(*
SPDX-FileCopyrightText: © 2026 Oleksandr Tiutyk <trofimich@gmail.com>
SPDX-License-Identifier: MIT
License: https://opensource.org/license/mit
*)

(*!
<summary>Exposes the compiler-initialized namespace of the Core library.</summary>
<description>Static internal storage; Name is a borrowed read-only view and requires no cyclic execution.</description>
*)

{attribute 'no_explicit_call' := 'do not call this POU directly'}
PROGRAM INTERNAL CurrentNamespace
VAR
	{attribute 'hide'} 
	_NamespaceExtractor : NamespaceExtractor;
END_VAR

(*!
<summary>Returns the compiler-initialized library namespace.</summary>
<description>Borrowed read-only reference to static storage. Do not modify it through the reference.</description>
*)
{attribute 'monitoring' := 'call'}
PROPERTY Name : REFERENCE TO STRING
GET
Name REF= _NamespaceExtractor.CurrentNamespace;
END_GET
END_PROPERTY

END_PROGRAM

(* stored: Version 1.1.0.1
   POU CurrentNamespace: Id {d326d085-4c96-43f5-a212-89329b4d09f9}, SpecialFunc None
   Property Name: Id {8f04ec1a-926d-4d00-b5c9-a6ab7edcc246}
   Get Get: Id {1a5a14b1-e1b1-4028-ad25-6a65e10c43cf} *)
